(* IEC 61131-3 sources: Industry-PLC-LLM/data/PLCBEAD_repo/PLCBEAD_PLCEmbed-main/PLC-BEAD/Source/GEB/TIME_TO_UDINT, 1 file *)

(* ---- TIME_TO_UDINT.ST ---- *)
FUNCTION TIME_TO_UDINT2:UDINT
	VAR_INPUT
		X :	TIME;
	END_VAR

	TIME_TO_UDINT2 := DINT_TO_UDINT(TIME_TO_DINT(X));
END_FUNCTION

PROGRAM program0
  VAR
    LocalVar0 : TIME;
    LocalOUT  : UDINT;
  END_VAR

  LocalOUT := TIME_TO_UDINT2(LocalVar0);
END_PROGRAM
